// Mitsubishi GX Developer project: traffic   PLC: FX3U

PROGRAM MAIN
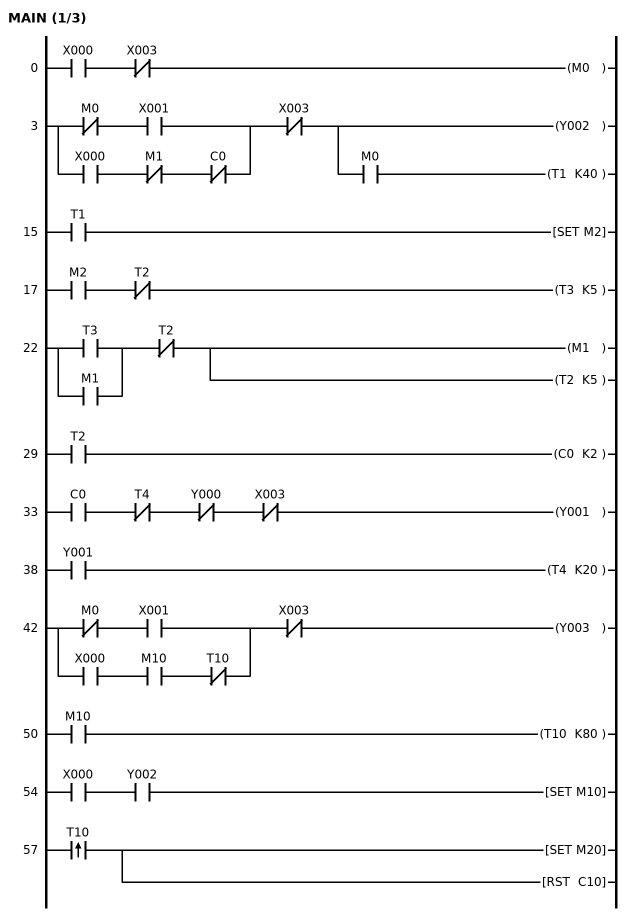
0     LD      X000
      ANI     X003
      OUT     M0
3     LDI     M0
      AND     X001
      LD      X000
      ANI     M1
      ANI     C0
      ORB
      ANI     X003
      OUT     Y002
      AND     M0
      OUT     T1 K40
15    LD      T1
      SET     M2
17    LD      M2
      ANI     T2
      OUT     T3 K5
22    LD      T3
      OR      M1
      ANI     T2
      OUT     M1
      OUT     T2 K5
29    LD      T2
      OUT     C0 K2
33    LD      C0
      ANI     T4
      ANI     Y000
      ANI     X003
      OUT     Y001
38    LD      Y001
      OUT     T4 K20
42    LDI     M0
      AND     X001
      LD      X000
      AND     M10
      ANI     T10
      ORB
      ANI     X003
      OUT     Y003
50    LD      M10
      OUT     T10 K80
54    LD      X000
      AND     Y002
      SET     M10
57    LDP     T10
      SET     M20
      RST     C10
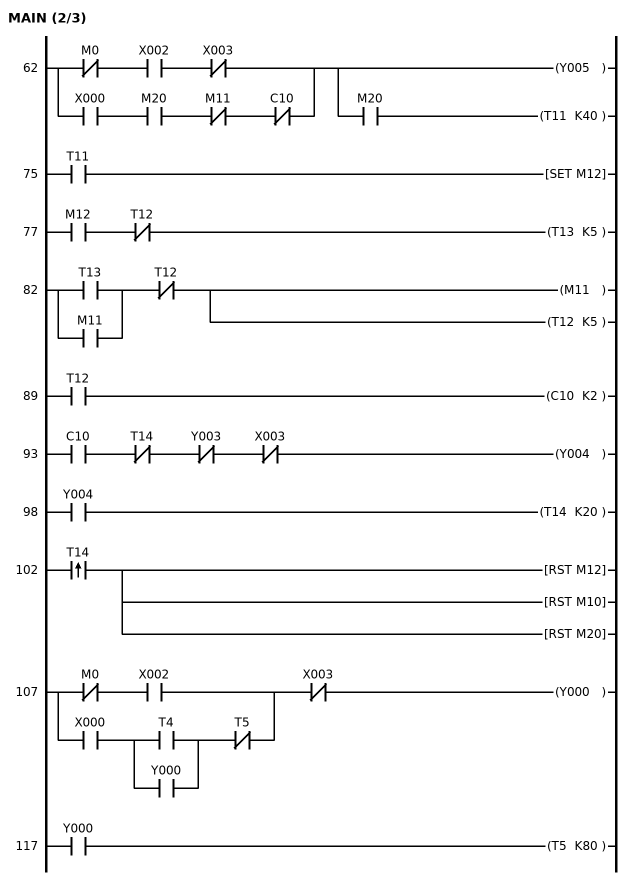
62    LDI     M0
      AND     X002
      ANI     X003
      LD      X000
      AND     M20
      ANI     M11
      ANI     C10
      ORB
      OUT     Y005
      AND     M20
      OUT     T11 K40
75    LD      T11
      SET     M12
77    LD      M12
      ANI     T12
      OUT     T13 K5
82    LD      T13
      OR      M11
      ANI     T12
      OUT     M11
      OUT     T12 K5
89    LD      T12
      OUT     C10 K2
93    LD      C10
      ANI     T14
      ANI     Y003
      ANI     X003
      OUT     Y004
98    LD      Y004
      OUT     T14 K20
102   LDP     T14
      RST     M12
      RST     M10
      RST     M20
107   LDI     M0
      AND     X002
      LD      X000
      LD      T4
      OR      Y000
      ANB
      ANI     T5
      ORB
      ANI     X003
      OUT     Y000
117   LD      Y000
      OUT     T5 K80
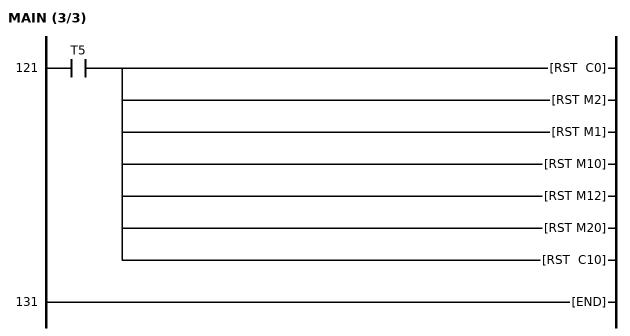
121   LD      T5
      RST     C0
      RST     M2
      RST     M1
      RST     M10
      RST     M12
      RST     M20
      RST     C10
131   END
END_PROGRAM
